Omron CX-Programmer project NewProject (CX-Programmer 9.77)

# PLC NewPLC1: CP1L-E EL

## Program NewProgram1 (cyclic task 0)

### Section Section1

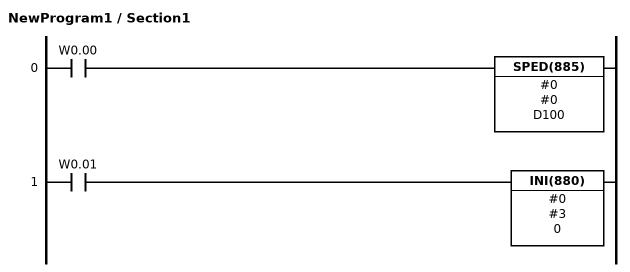
; rung 0
LD W0.00
SPED(885) #0 #0 D100
; rung 1
LD W0.01
INI(880) #0 #3 0
; rung 2
END(001)